(* Schneider Machine Expert - Basic project Running LED, file version 1.7.0.0 *)
(* ProjectInformations: Name=New project *)

HARDWARE
  Cpu 0: TM221M16R/G
  EthernetConfiguration: NetworkName=M221, IpAllocationMode=FixedAddress, IpAddress=0.0.0.0, SubnetMask=0.0.0.0
  SerialLineConfiguration: Baud=Baud19200, Parity=ParityEven, DataBits=DataBits8, StopBits=StopBits1, PhysicalMedium=PhysicalMediumRs485, TransmissionMode=TransmissionModeModbusRtu, SlaveId=1, Addressing=SlaveAddressing
  MastTask: UsePeriodScanMode=false, PeriodScan=100
  FastTask: Period=255
  CpuBehavior: StartingMode=StartAsPreviousState, AutoSaveRamOnEeprom=true, WatchdogPeriod=250

SYMBOLS  (address, symbol, comment, settings)
  %TM1        [Preset=1, Base=OneSecond]
  %TM2        [Preset=1, Base=OneSecond]
  %TM3        [Preset=1, Base=OneSecond]
  %TM4        [Preset=1, Base=OneSecond]
  %TM5        [Preset=1, Base=OneSecond]
  %TM6        [Preset=1, Base=OneSecond]
  %TM7        [Preset=1, Base=OneSecond]
  %TM8        [Preset=1, Base=OneSecond]

POU New POU
  (* SectionNumber=1 *)

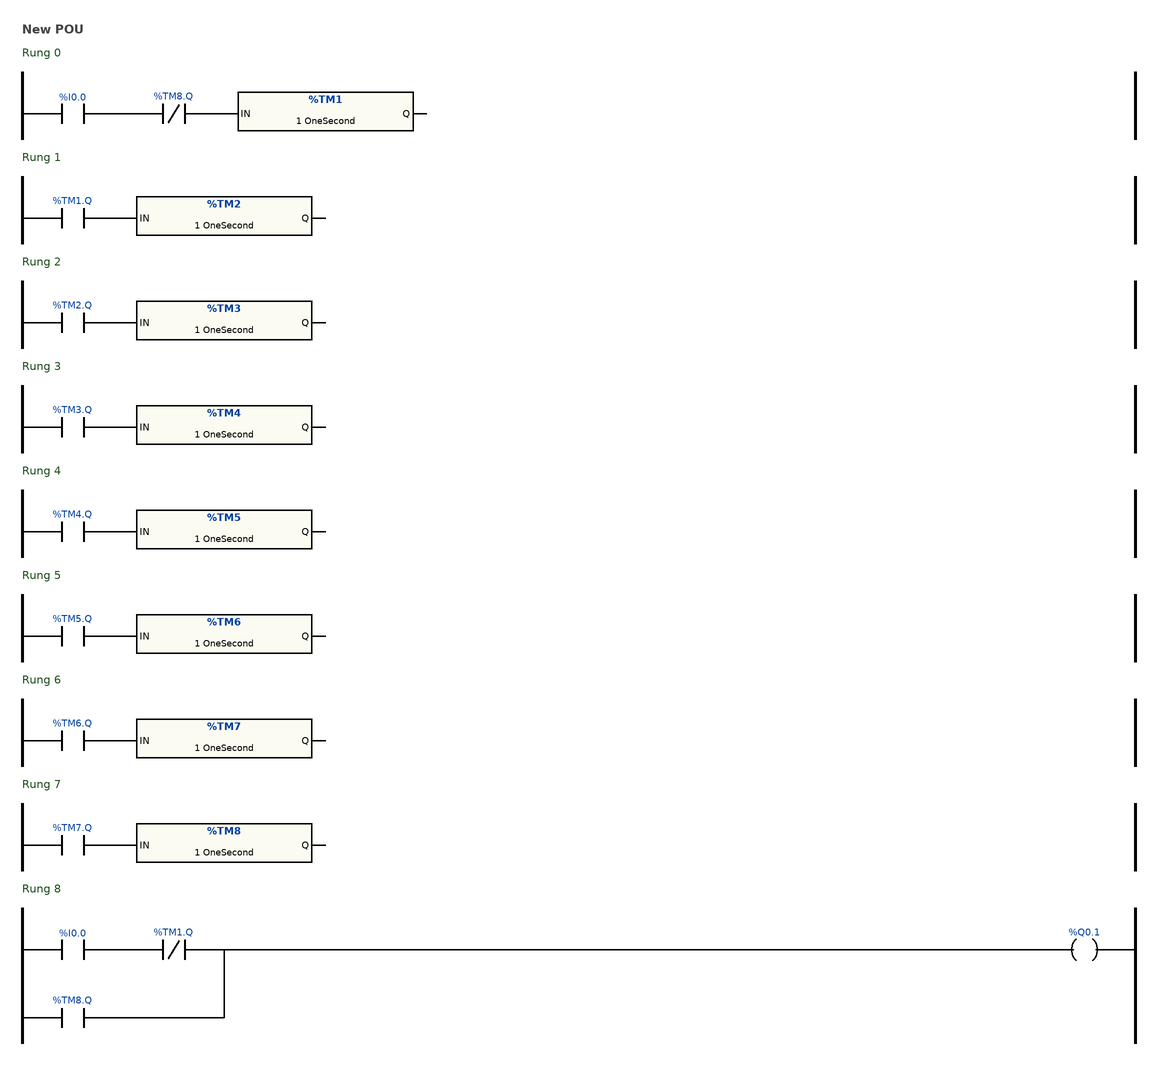

// Rung 0
  BLK %TM1
  LD %I0.0
  ANDN %TM8.Q
  IN
  END_BLK
  // as ST:
  //   %TM1(IN := %I0.0 AND NOT %TM8.Q);

// Rung 1
  BLK %TM2
  LD %TM1.Q
  IN
  END_BLK
  // as ST:
  //   %TM2(IN := %TM1.Q);

// Rung 2
  BLK %TM3
  LD %TM2.Q
  IN
  END_BLK
  // as ST:
  //   %TM3(IN := %TM2.Q);

// Rung 3
  BLK %TM4
  LD %TM3.Q
  IN
  END_BLK
  // as ST:
  //   %TM4(IN := %TM3.Q);

// Rung 4
  BLK %TM5
  LD %TM4.Q
  IN
  END_BLK
  // as ST:
  //   %TM5(IN := %TM4.Q);

// Rung 5
  BLK %TM6
  LD %TM5.Q
  IN
  END_BLK
  // as ST:
  //   %TM6(IN := %TM5.Q);

// Rung 6
  BLK %TM7
  LD %TM6.Q
  IN
  END_BLK
  // as ST:
  //   %TM7(IN := %TM6.Q);

// Rung 7
  BLK %TM8
  LD %TM7.Q
  IN
  END_BLK
  // as ST:
  //   %TM8(IN := %TM7.Q);

// Rung 8
  LD %I0.0
  ANDN %TM1.Q
  OR %TM8.Q
  ST %Q0.1
  // as ST:
  //   %Q0.1 := %I0.0 AND NOT %TM1.Q OR %TM8.Q;

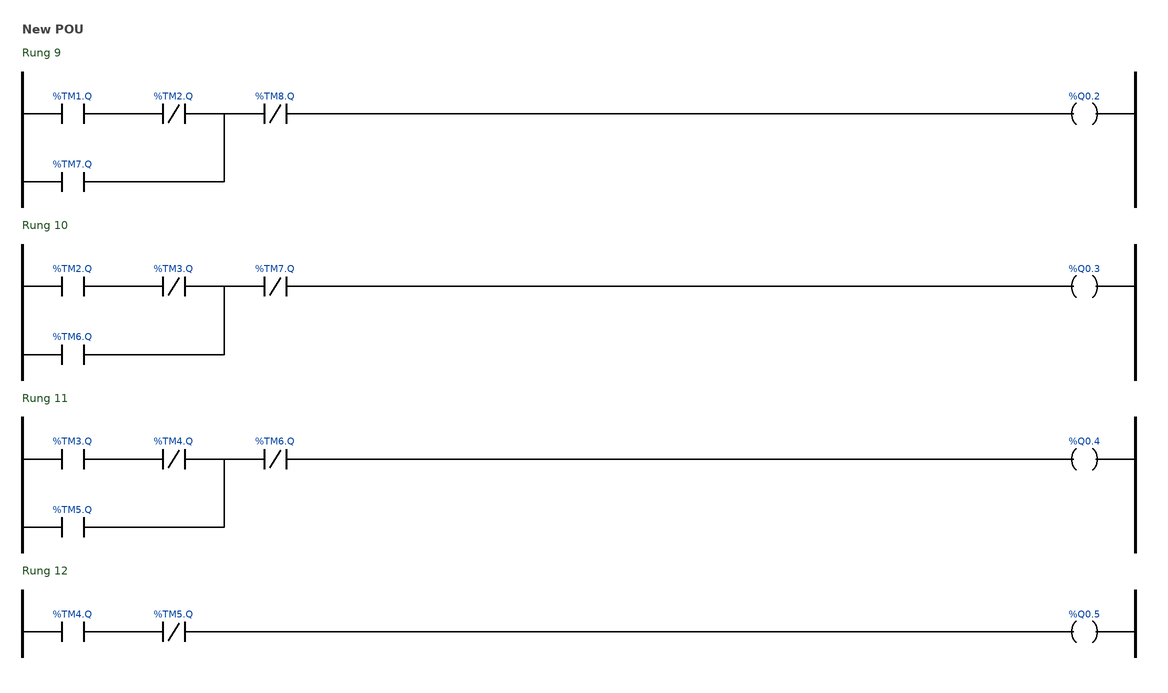

// Rung 9
  LD %TM1.Q
  ANDN %TM2.Q
  OR %TM7.Q
  ANDN %TM8.Q
  ST %Q0.2
  // as ST:
  //   %Q0.2 := (%TM1.Q AND NOT %TM2.Q OR %TM7.Q) AND NOT %TM8.Q;

// Rung 10
  LD %TM2.Q
  ANDN %TM3.Q
  OR %TM6.Q
  ANDN %TM7.Q
  ST %Q0.3
  // as ST:
  //   %Q0.3 := (%TM2.Q AND NOT %TM3.Q OR %TM6.Q) AND NOT %TM7.Q;

// Rung 11
  LD %TM3.Q
  ANDN %TM4.Q
  OR %TM5.Q
  ANDN %TM6.Q
  ST %Q0.4
  // as ST:
  //   %Q0.4 := (%TM3.Q AND NOT %TM4.Q OR %TM5.Q) AND NOT %TM6.Q;

// Rung 12
  LD %TM4.Q
  ANDN %TM5.Q
  ST %Q0.5
  // as ST:
  //   %Q0.5 := %TM4.Q AND NOT %TM5.Q;
